FUNCTION_BLOCK Test_ExampleTest EXTENDS T_UnitTestBase

METHOD RunTest
VAR
    TestValue : LREAL := 133.456;
END_VAR
AssertEquals_LREAL(Expected := 133.456,
                    Actual   := TestValue,
                    Delta    := 0.001,
                    Message  := 'TestValue <> 133.456');

TestCompleted := TRUE;
END_METHOD

END_FUNCTION_BLOCK

(* stored: Version 1.1.0.1, ProductVersion 3.1.4024.12
   POU Test_ExampleTest: Id {938982c1-236f-47a0-9361-5ca61f22a12c}, SpecialFunc None
   Method RunTest: Id {d43fbc30-af37-40f9-89b6-ca71e886dbd4} *)
